// Brief: Slave Arm Invase instrument to record position
FUNCTION_BLOCK PUBLIC FB_SlaveCtrlInstruInvasion EXTENDS FB_SlaveArmCtrlBase
VAR_INPUT
END_VAR
VAR_OUTPUT
END_VAR
VAR
	// invasion buffer
	m_instruInvasionDepthSafetyBuffer :LREAL:= 0.01;
		
	// max damping when reaching invasion depth
	m_maxDamp :LREAL :=100;
	
	// current distance form target invasion depth 
	m_invasionDis :LREAL :=0;
	
	// distance threshold from target depth to start enable damp
	m_dampDisThres :LREAL :=0.03;
	
	// velocity for full damping
	m_maxAdjustVel :LREAL := 0.3;
	
	// velocity start to enable damping
	m_velLBForDamp :LREAL := 0.2;
	
END_VAR

// override this function in each exact controller
METHOD PROTECTED calcCmdJntPos : BOOL
VAR_IN_OUT CONSTANT
	i_endoscopePose : ST_Frame;
	i_masterStatus :ST_MasterStatus;
	i_setupStatus: ST_SetupStatus;
	i_slaveArm :FB_SlaveArm;
END_VAR

VAR 
	curInstruDepth:LREAL;
END_VAR
m_cmdJntPos[3]:=i_slaveArm.curJntPos[3];
// compute current instrument depth
curInstruDepth := i_slaveArm.curJntPos[3]-i_slaveArm.instrument.instruTypeInfo.m_rodLength-i_slaveArm.instrument.instruTypeInfo.m_headLength
						- i_slaveArm.instrument.instruTypeInfo.m_fingerLength-m_instruInvasionDepthSafetyBuffer;

m_invasionDis:=curInstruDepth-i_slaveArm.m_instruInvasionDepth;
						
m_isFinished := curInstruDepth<= i_slaveArm.m_instruInvasionDepth;
END_METHOD

// override this function in each exact controller
METHOD PROTECTED calcCmdJntTrq : BOOL
VAR_IN_OUT CONSTANT
	i_endoscopePose : ST_Frame;
	i_masterStatus :ST_MasterStatus;
	i_setupStatus: ST_SetupStatus;
	i_slaveArm :FB_SlaveArm;
END_VAR
VAR
	dampScale :lreal ;
END_VAR
// set joint torque to zero in default
m_cmdJntTrq := g_zeroVec8d;
		
// postion damp
dampScale  :=LIMIT(0, 1-m_invasionDis/m_dampDisThres,1);
m_cmdJntTrq[3]:= -dampScale * m_maxDamp * i_slaveArm.curJntVel[3];

// velocity damp
dampScale:=LIMIT(0, (ABS(i_slaveArm.curJntVel[3])- m_velLBForDamp)/(m_maxAdjustVel - m_velLBForDamp), 1 );
m_cmdJntTrq[3] :=m_cmdJntTrq[3] -i_slaveArm.curJntVel[3] * m_maxDamp * dampScale;
END_METHOD

METHOD PUBLIC init : BOOL
VAR_IN_OUT CONSTANT
	i_slaveArm	:FB_SlaveArm;
END_VAR
VAR_IN_OUT 
	r_slaveArmCtrlCmd :ST_SlaveArmCtrlCmds;
END_VAR
// check if to hold the command joint position unchanged
m_holdLastCmds := checkToHoldLastCmds(i_slaveArm);

//init
SUPER^.Init(i_slaveArm,r_slaveArmCtrlCmd);
m_invasionDis:=m_dampDisThres;

// only joint 3 is allowed to be pushed
m_jntOPMode := g_slaveAllPosTrqMode;
m_jntOPMode[3]:=DriverOPMode_Trq;

// update commands to arm
copyCmds(r_slaveArmCtrlCmd);

//check instrument type, DepthSafetyBuffer = 0 if instrument type is endoscope
IF i_slaveArm.instrument.instruType = InstruType_Endoscope THEN
	m_instruInvasionDepthSafetyBuffer := 0 ;
ELSE
	m_instruInvasionDepthSafetyBuffer := 0.010;
END_IF
END_METHOD

END_FUNCTION_BLOCK

(* stored: Version 1.1.0.1, ProductVersion 3.1.4024.11
   POU FB_SlaveCtrlInstruInvasion: Id {ea7b020b-d76c-4bb7-93d3-7a449a773602}, SpecialFunc None
   Method calcCmdJntPos: Id {69de60b3-1c13-41f6-898e-63d0fb34a945}
   Method calcCmdJntTrq: Id {48bb9834-7afe-4e4a-9ec9-117889c76c2c}
   Method init: Id {bcdf683e-60d5-4385-b995-2cd1f6e8f528} *)
